SUBAPPLICATION Uebung_071b (* WBSD auf UT ausgeben, Q1 Schalten wenn Speed &gt;0 *)
  (* Standard: 61499-2 *)
  (* Version 1.0, 2023-10-23, franz *)
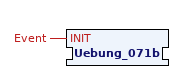
  EVENT_INPUT
    INIT;
  END_EVENT
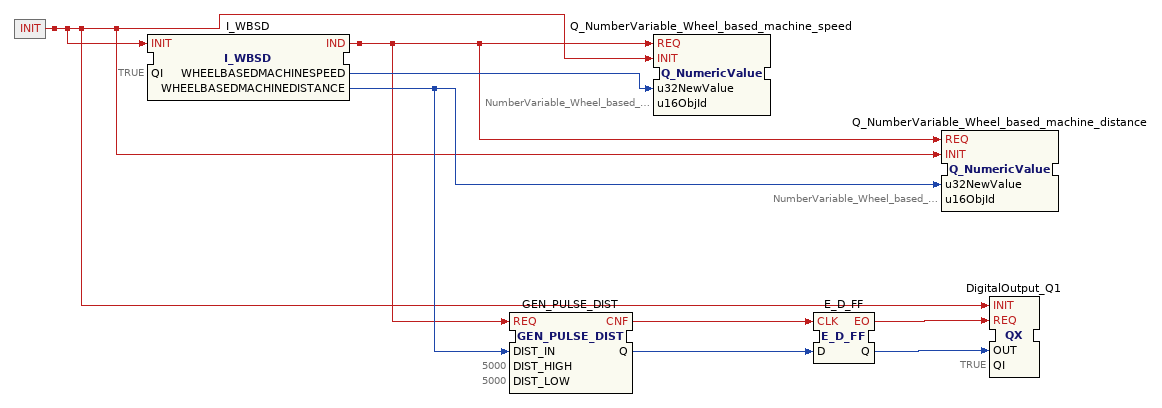
  FBS
    I_WBSD : I_WBSD(QI := TRUE);
    Q_NumberVariable_Wheel_based_machine_speed : Q_NumericValue(u16ObjId := NumberVariable_Wheel_based_machine_speed);
    DigitalOutput_Q1 : QX(QI := TRUE);
    GEN_PULSE_DIST : signalprocessing::distance::GEN_PULSE_DIST(DIST_HIGH := 5000, DIST_LOW := 5000);
    E_D_FF : E_D_FF;
    Q_NumberVariable_Wheel_based_machine_distance : Q_NumericValue(u16ObjId := NumberVariable_Wheel_based_machine_distance);
  END_FBS
  EVENT_CONNECTIONS
    I_WBSD.IND TO Q_NumberVariable_Wheel_based_machine_speed.REQ;
    INIT TO I_WBSD.INIT;
    INIT TO Q_NumberVariable_Wheel_based_machine_speed.INIT;
    INIT TO DigitalOutput_Q1.INIT;
    I_WBSD.IND TO GEN_PULSE_DIST.REQ;
    E_D_FF.EO TO DigitalOutput_Q1.REQ;
    GEN_PULSE_DIST.CNF TO E_D_FF.CLK;
    I_WBSD.IND TO Q_NumberVariable_Wheel_based_machine_distance.REQ;
    INIT TO Q_NumberVariable_Wheel_based_machine_distance.INIT;
  END_CONNECTIONS
  DATA_CONNECTIONS
    I_WBSD.WHEELBASEDMACHINESPEED TO Q_NumberVariable_Wheel_based_machine_speed.u32NewValue;
    I_WBSD.WHEELBASEDMACHINEDISTANCE TO GEN_PULSE_DIST.DIST_IN;
    E_D_FF.Q TO DigitalOutput_Q1.OUT;
    GEN_PULSE_DIST.Q TO E_D_FF.D;
    I_WBSD.WHEELBASEDMACHINEDISTANCE TO Q_NumberVariable_Wheel_based_machine_distance.u32NewValue;
  END_CONNECTIONS
END_SUBAPPLICATION
